Staubli VAL3: chkAtHome.pgx

program chkAtHome(bool& x_bIsHome)
begin
  //判读机器人是否在安全位置
  if abs(PublicData:jHome)<{0.1,0.1,0.1,0.1,0.1,0.1}
    popUpMsg("机器人安全位置：6个轴都不能为零.")
    x_bIsHome=false
    return
  endIf

  if abs(herej()-PublicData:jHome)>{0.1,0.1,0.1,0.1,0.1,0.1}
    x_bIsHome=false
    popUpMsg("机器人不在安全位置。")
  else
    x_bIsHome=true
  endIf
end
